// TIA Portal V17 export
// export: Created 2023-07-20T16:54:09.7783395Z, ExportSetting WithDefaults, DisplayName Totally Integrated Automation Portal, DisplayVersion V17, DisplayName TIA Portal Openness, DisplayVersion V17, DisplayName TIA Portal Version Control Interface, DisplayVersion V17, DisplayName STEP 7 Professional, DisplayVersion V17, DisplayName STEP 7 Safety, DisplayVersion V17, DisplayName WinCC Professional, DisplayVersion V17
FUNCTION "Modbus RTU handler" : Void   // FC10, LAD
TITLE = Modbus RTU handler
{ S7_Optimized_Access := 'TRUE' }
VERSION : 0.1
// This block updates R/W data from all the devices connected to the designated CM 1241 module.
// 
// Peripherals connected to this module:
// 
// -AZD-KD
// stored: AutoNumber false, IsIECCheckEnabled false, SetENOAutomatically false, UDAEnableTagReadback false
BEGIN

REGION Network 1: Modbus RTU module setup block
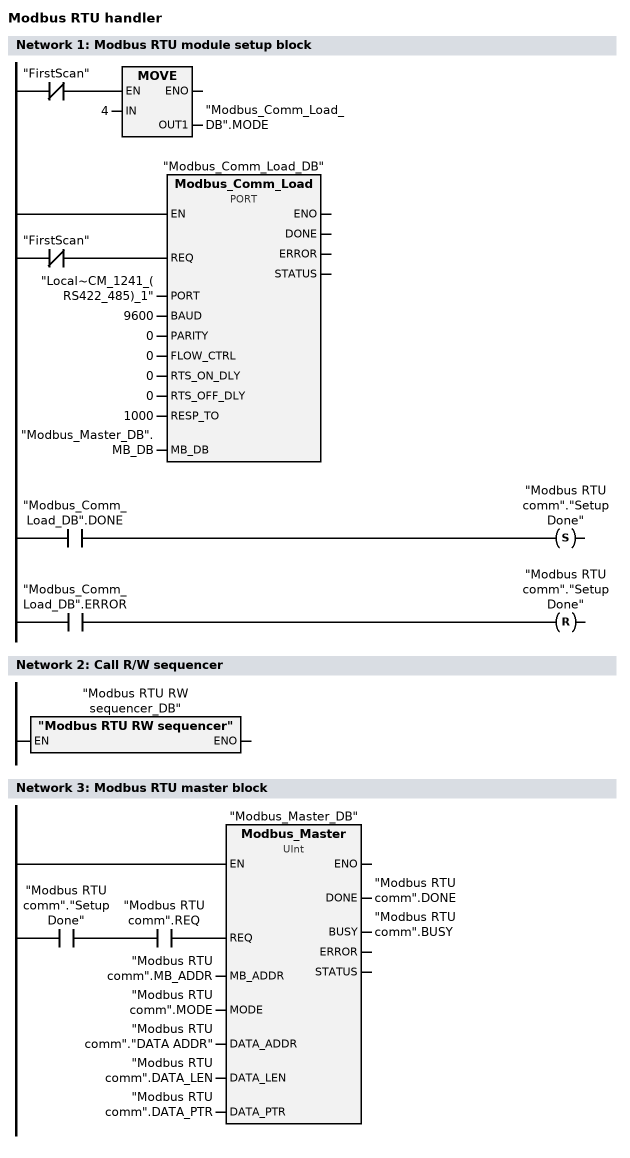
   RUNG wire#powerrail
      I_Contact( "FirstScan" )
      Move(in := 4, out1 => "Modbus_Comm_Load_DB".MODE)
   END_RUNG
   RUNG wire#powerrail
      { S7_Templates := "[card := 0, port_type := PORT, word_type := UInt, dint_type := UDInt, mbbase_type := P2P_MB_BASE]" } "Modbus_Comm_Load_DB".Modbus_Comm_Load(REQ := wire#w1, PORT := "Local~CM_1241_(RS422_485)_1", BAUD := 9600, PARITY := 0, FLOW_CTRL := 0, RTS_ON_DLY := 0, RTS_OFF_DLY := 0, RESP_TO := 1000, MB_DB := "Modbus_Master_DB".MB_DB, DONE =>, ERROR =>, STATUS =>)
   END_RUNG
   RUNG wire#powerrail
      I_Contact( "FirstScan" )
   END_RUNG wire#w1
   RUNG wire#powerrail
      Contact( "Modbus_Comm_Load_DB".DONE )
      S_Coil( "Modbus RTU comm"."Setup Done" )
   END_RUNG
   RUNG wire#powerrail
      Contact( "Modbus_Comm_Load_DB".ERROR )
      R_Coil( "Modbus RTU comm"."Setup Done" )
   END_RUNG
   // the same network as SCL:
   IF NOT "FirstScan" THEN "Modbus_Comm_Load_DB".MODE := 4; END_IF;
   "Modbus_Comm_Load_DB"(REQ := NOT "FirstScan",   // Modbus_Comm_Load
                         PORT := "Local~CM_1241_(RS422_485)_1",
                         BAUD := 9600,
                         PARITY := 0,
                         FLOW_CTRL := 0,
                         RTS_ON_DLY := 0,
                         RTS_OFF_DLY := 0,
                         RESP_TO := 1000,
                         MB_DB := "Modbus_Master_DB".MB_DB);
   IF "Modbus_Comm_Load_DB".DONE THEN "Modbus RTU comm"."Setup Done" := TRUE; END_IF;
   IF "Modbus_Comm_Load_DB".ERROR THEN "Modbus RTU comm"."Setup Done" := FALSE; END_IF;
END_REGION

REGION Network 2: Call R/W sequencer
   RUNG wire#powerrail
      "Modbus RTU RW sequencer_DB"()
   END_RUNG
   // the same network as SCL:
   "Modbus RTU RW sequencer_DB"();   // "Modbus RTU RW sequencer"
END_REGION

REGION Network 3: Modbus RTU master block
   RUNG wire#powerrail
      { S7_Templates := "[card := 0, word_type := UInt, dword_type := UDInt, byte_type := USInt, any_type := Variant]" } "Modbus_Master_DB".Modbus_Master(REQ := wire#w1, MB_ADDR := "Modbus RTU comm".MB_ADDR, MODE := "Modbus RTU comm".MODE, DATA_ADDR := "Modbus RTU comm"."DATA ADDR", DATA_LEN := "Modbus RTU comm".DATA_LEN, DATA_PTR := "Modbus RTU comm".DATA_PTR, DONE => "Modbus RTU comm".DONE, BUSY => "Modbus RTU comm".BUSY, ERROR =>, STATUS =>)
   END_RUNG
   RUNG wire#powerrail
      Contact( "Modbus RTU comm"."Setup Done" )
      Contact( "Modbus RTU comm".REQ )
   END_RUNG wire#w1
   // the same network as SCL:
   "Modbus_Master_DB"(REQ := "Modbus RTU comm"."Setup Done" AND "Modbus RTU comm".REQ,   // Modbus_Master
                      MB_ADDR := "Modbus RTU comm".MB_ADDR,
                      MODE := "Modbus RTU comm".MODE,
                      DATA_ADDR := "Modbus RTU comm"."DATA ADDR",
                      DATA_LEN := "Modbus RTU comm".DATA_LEN,
                      DATA_PTR := "Modbus RTU comm".DATA_PTR,
                      DONE => "Modbus RTU comm".DONE,
                      BUSY => "Modbus RTU comm".BUSY);
END_REGION
END_FUNCTION
